	!Check that there are no more than 3 numbers in the signal description
	WHILE n_CharNumberCount>2 DO
		TPErase;
		st_MsgBoxHeader:=["GetGOValue  Signal=" + st_doSignalName ,"GetGOValue  Signal=" + st_doSignalName,"???"];
		st_MsgBoxLine3:=["There are more than two numbers in the" ,"Es gibt mehr als zwei Zahlen in der","???"];
		st_MsgBoxLine4:=["signal name defined. Check Configuration.","Signal-Name definiert. Konfiguration prüfen.","???"];
		n_MsgBoxAnswer:= UIMessageBox (\Header:=st_MsgBoxHeader{n_Sp}\MsgArray:=[" "," ",st_MsgBoxLine3{n_Sp},st_MsgBoxLine4{n_Sp}," "]\Buttons:=btnOK\Icon:=iconError) ;

		STOP;
	ENDWHILE

	!Check that there are no less than numbers in signal description
	WHILE n_CharNumberCount<2 DO
		TPErase;
		st_MsgBoxHeader:=["GetGOValue  Signal=" + st_doSignalName ,"GetGOValue  Signal=" + st_doSignalName,"???"];
		st_MsgBoxLine3:=["The are less than two numbers in the" ,"???","???"];
		st_MsgBoxLine4:=["signal name defined. Check Configuration.","Signal-Name definiert. Konfiguration prüfen.","???"];
		n_MsgBoxAnswer:= UIMessageBox (\Header:=st_MsgBoxHeader{n_Sp}\MsgArray:=[" "," ",st_MsgBoxLine3{n_Sp},st_MsgBoxLine4{n_Sp}," "]\Buttons:=btnOK\Icon:=iconError) ;

		STOP;
	ENDWHILE

	!Get Bit number as a string
	st_FirstbitNr:=StrPart(st_doSignalName,n_CharFirstNumber,n_NumberCharlength);

	!Check st_FirstbitNr is a number
	WHILE StrToVal(st_FirstbitNr,n_FirstBitNr)<>TRUE DO
		TPErase;
		st_MsgBoxHeader:=["GetGOValue  Signal=" + st_doSignalName ,"GetGOValue  Signal=" + st_doSignalName,"???"];
		st_MsgBoxLine3:=["There are not two consecutive bit numbers defined." ,"Es gibt nicht zwei aufeinander folgenden Bit-Zahlen definiert.","???"];
		st_MsgBoxLine4:=["Please Check Configuration.","Bitte Überprüfe Konfiguration.","???"];
		n_MsgBoxAnswer:= UIMessageBox (\Header:=st_MsgBoxHeader{n_Sp}\MsgArray:=[" "," ",st_MsgBoxLine3{n_Sp},st_MsgBoxLine4{n_Sp}," "]\Buttons:=btnOK\Icon:=iconError) ;

		STOP;
	ENDWHILE

	st_doSignalDesc1:=StrPart(st_doSignalName,1,n_CharFirstNumber-1);

	IF (n_CharFirstNumber+1)=n_doSignal_Length OR n_CharFirstNumber=n_doSignal_Length THEN
		!Bit numbers are the last two characters
		st_doSignalDesc2:="" ;
		st_doSignalDesc:=st_doSignalDesc1 + "??" ;
	ELSE
		st_doSignalDesc2:=StrPart(st_doSignalName,n_CharFirstNumber+2,n_doSignal_Length-n_CharFirstNumber-1);
		st_doSignalDesc:=st_doSignalDesc1 + "??" + st_doSignalDesc2 ;
	ENDIF

	n_LastBitNr:=n_FirstBitNr+n_doBitLength-1;

	IF n_doBitLength<1 OR n_doBitLength>16 THEN
		!Check n_doBitLength paramater is valid

		WHILE TRUE DO
			TPErase;
			st_MsgBoxHeader:=["GetGOValue  Signal=" + st_doSignalName ,"GetGOValue  Signal=" + st_doSignalName,"???"];
			st_MsgBoxLine3:=["The Bit length Specified=" + ValToStr(n_doBitLength) + ". Value must be between 1-16." ,"Die Bitlänge angegeben=" + ValToStr(n_doBitLength) + ". Wert muss zwischen 1-16.","???"];
			st_MsgBoxLine4:=["Please Check Configuration.","Bitte Überprüfe Konfiguration.","???"];
			n_MsgBoxAnswer:= UIMessageBox (\Header:=st_MsgBoxHeader{n_Sp}\MsgArray:=[" "," ",st_MsgBoxLine3{n_Sp},st_MsgBoxLine4{n_Sp}," "]\Buttons:=btnOK\Icon:=iconError) ;

			STOP;
		ENDWHILE

	ELSEIF n_LastBitNr>32 THEN
		!Check last bit number

		WHILE TRUE DO
			TPErase;
			st_MsgBoxHeader:=["GetGOValue  Signal=" + st_doSignalName ,"GetGOValue  Signal=" + st_doSignalName,"???"];
			st_MsgBoxLine3:=["The first Bit specified=" + ValToStr(n_FirstBitNr) + " + length specified=" + ValToStr(n_doBitLength) + " is >32.","Die Erstes Bit angegeben=" + ValToStr(n_FirstBitNr) + " + Länge angegeben=" + ValToStr(n_doBitLength) + " ist >32.","???"];
			st_MsgBoxLine4:=["Please Check Configuration.","Bitte Überprüfe Konfiguration.","???"];
			n_MsgBoxAnswer:= UIMessageBox (\Header:=st_MsgBoxHeader{n_Sp}\MsgArray:=[" "," ",st_MsgBoxLine3{n_Sp},st_MsgBoxLine4{n_Sp}," "]\Buttons:=btnOK\Icon:=iconError) ;

			STOP;
		ENDWHILE

	ELSE !n_doBitLength<1
		n_ScrollNr:=0.5;
		n_ValueCount:=0;

		FOR n_CharNr FROM n_FirstBitNr	TO n_LastBitNr DO
			n_ScrollNr:=n_ScrollNr*2;

			IF n_CharNr<10 AND n_CharFirstNumber<>n_doSignal_Length THEN
				st_tempString:=st_doSignalDesc1 +"0" + ValToStr(n_CharNr) + st_doSignalDesc2;
			ELSE
				st_tempString:=st_doSignalDesc1 + ValToStr(n_CharNr) + st_doSignalDesc2;
			ENDIF

			AliasIO st_tempString, do_Temp;

			IF doutput(do_Temp) = 1 THEN
				n_ValueCount:=n_ValueCount + n_ScrollNr ;
			ENDIF

		ENDFOR

		n_LastGroupOutput:=n_ValueCount;
		RETURN n_ValueCount ;
	ENDIF !n_doBitLength<1
ENDIF !n_diSignal_Length

ERROR
!** Error Handler **

TEST  ERRNO
CASE ERR_ALIASIO_DEF,ERR_ALIASIO_TYPE :
	WHILE TRUE DO
		TPErase;
		st_MsgBoxHeader:=["GetGOValue Signal=" + st_tempString ,"GetGOValue Signal=" + st_tempString,"???"];
		st_MsgBoxLine3:=["Signal is missing or incorrectly defined","IO Signal ist nicht vorhanden oder Falsch geschrieben","???"];
		st_MsgBoxLine4:=["Please Check Configuration.","Bitte Überprüfe Konfiguration.","???"];
		n_MsgBoxAnswer:= UIMessageBox (\Header:=st_MsgBoxHeader{n_Sp}\MsgArray:=[" "," ",st_MsgBoxLine3{n_Sp},st_MsgBoxLine4{n_Sp}," "]\Buttons:=btnOK\Icon:=iconError) ;

		STOP;
	ENDWHILE
DEFAULT :
	WHILE TRUE DO
		TPErase;
		st_MsgBoxHeader:=["GetGOValue Unknown Error =" + ValToStr(Errno) ,"GetGOValue unbekannter Fehler =" + ValToStr(Errno),"???"];
		st_MsgBoxLine3:=["Support Required.","Unterstützung erforderlich.","???"];
		st_MsgBoxLine4:=[" "," ","???"];
		n_MsgBoxAnswer:= UIMessageBox (\Header:=st_MsgBoxHeader{n_Sp}\MsgArray:=[" "," ",st_MsgBoxLine3{n_Sp},st_MsgBoxLine4{n_Sp}," "]\Buttons:=btnOK\Icon:=iconError) ;

		STOP;
	ENDWHILE
ENDTEST

ENDFUNC !(GetGroupOP)


!*******************************************************************************


PROC SetGroupOP (VAR Signaldo doSignalName,Num n_doBitLength,Num n_doSetValue)
!************************************
!* Procedure set a group of Digital *
!* Outputs based on a numeric value *
!************************************

VAR signaldo do_Temp;

VAR Byte by_HighByte ;
VAR Byte by_LowByte ;
VAR Byte by_BitMask;

VAR Num n_FirstBitNr;
VAR Num n_LastBitNr;
VAR Num n_doSignal_Length;
VAR Num n_CharNr;
VAR Num n_ScrollNr;
VAR Num n_CharFirstNumber;
VAR Num n_CharNumberCount;
VAR Num n_MaxValue ;
VAR Num n_TempNr ;
VAR Num n_ChkValue ;
VAR Num n_TempDoValue ;

VAR String st_doSignalName;
VAR String st_FirstbitNr;
VAR String st_doSignalDesc;
VAR String st_doSignalDesc1;
VAR String st_doSignalDesc2;
VAR String st_tempString ;

!Stop advance pointer
WaitTime\Inpos, 0.0 ;

!Check first bit configured is a valid output
st_doSignalName:=ArgName(doSignalName);
AliasIO st_doSignalName, do_Temp;

!Check output name length
n_doSignal_Length:=StrLen(st_doSignalName);

IF n_doSignal_Length > 3 THEN
	!Determine which characters the Bit numbers start
	n_CharFirstNumber:=StrFind(st_doSignalName,1,STR_DIGIT) ;

	!Check that there are numbers in signal description
	WHILE n_CharFirstNumber>n_doSignal_Length DO
		TPErase;
		st_MsgBoxHeader:=["SetGOValue Signal=" + st_doSignalName ,"SetGOValue Signal=" + st_doSignalName,"???"];
		st_MsgBoxLine3:=["There are no bit numbers in the signal name defined." ,"Es gibt keine Bit-Zahlen in der Signal-Namen definiert","???"];
		st_MsgBoxLine4:=["Please Check Configuration.","Bitte Überprüfe Konfiguration.","???"];
		n_MsgBoxAnswer:= UIMessageBox (\Header:=st_MsgBoxHeader{n_Sp}\MsgArray:=[" "," ",st_MsgBoxLine3{n_Sp},st_MsgBoxLine4{n_Sp}," "]\Buttons:=btnOK\Icon:=iconError) ;

		STOP;
	ENDWHILE

	n_CharNumberCount:=1;

	!Check how many characters are numbers
	FOR n_CharNr FROM n_CharFirstNumber +1 TO n_doSignal_Length DO
		IF StrFind(st_doSignalName,n_CharNr,STR_DIGIT)<=n_doSignal_Length THEN
			INCR n_CharNumberCount ;
		ENDIF
	ENDFOR

	!Check that there are no more than 3 numbers in the signal description
	WHILE n_CharNumberCount>2 DO
		TPErase;
		st_MsgBoxHeader:=["SetGOValue Signal=" + st_doSignalName ,"SetGOValue Signal=" + st_doSignalName,"???"];
		st_MsgBoxLine3:=["There are more than two numbers in the" ,"Es gibt mehr als zwei Zahlen in der","???"];
		st_MsgBoxLine4:=["signal name defined. Check Configuration.","Signal-Name definiert. Konfiguration prüfen.","???"];
		n_MsgBoxAnswer:= UIMessageBox (\Header:=st_MsgBoxHeader{n_Sp}\MsgArray:=[" "," ",st_MsgBoxLine3{n_Sp},st_MsgBoxLine4{n_Sp}," "]\Buttons:=btnOK\Icon:=iconError) ;

		STOP;
	ENDWHILE

	!Check that there are no less than numbers in signal description
	WHILE n_CharNumberCount<2 DO
		TPErase;
		st_MsgBoxHeader:=["SetGOValue Signal=" + st_doSignalName ,"SetGOValue Signal=" + st_doSignalName,"???"];
		st_MsgBoxLine3:=["The are less than two numbers in the" ,"???","???"];
		st_MsgBoxLine4:=["signal name defined. Check Configuration.","Signal-Name definiert. Konfiguration prüfen.","???"];
		n_MsgBoxAnswer:= UIMessageBox (\Header:=st_MsgBoxHeader{n_Sp}\MsgArray:=[" "," ",st_MsgBoxLine3{n_Sp},st_MsgBoxLine4{n_Sp}," "]\Buttons:=btnOK\Icon:=iconError) ;

		STOP;
	ENDWHILE

	!Get Bit number as a string
	st_FirstbitNr:=StrPart(st_doSignalName,n_CharFirstNumber,2);

	!Check st_FirstbitNr is a number
	WHILE StrToVal(st_FirstbitNr,n_FirstBitNr)<>TRUE DO
		TPErase;
		st_MsgBoxHeader:=["SetGOValue Signal=" + st_doSignalName ,"SetGOValue Signal=" + st_doSignalName,"???"];
		st_MsgBoxLine3:=["There are not two consecutive bit numbers defined." ,"Es gibt nicht zwei aufeinander folgenden Bit-Zahlen definiert.","???"];
		st_MsgBoxLine4:=["Please Check Configuration.","Bitte Überprüfe Konfiguration.","???"];
		n_MsgBoxAnswer:= UIMessageBox (\Header:=st_MsgBoxHeader{n_Sp}\MsgArray:=[" "," ",st_MsgBoxLine3{n_Sp},st_MsgBoxLine4{n_Sp}," "]\Buttons:=btnOK\Icon:=iconError) ;

		STOP;
	ENDWHILE

	st_doSignalDesc1:=StrPart(st_doSignalName,1,n_CharFirstNumber-1);

	IF (n_CharFirstNumber+1)=n_doSignal_Length THEN
		!Bit numbers are the last two characters
		st_doSignalDesc2:="" ;
		st_doSignalDesc:=st_doSignalDesc1 + "??" ;
	ELSE
		st_doSignalDesc2:=StrPart(st_doSignalName,n_CharFirstNumber+2,n_doSignal_Length-n_CharFirstNumber-1);
		st_doSignalDesc:=st_doSignalDesc1 + "??" + st_doSignalDesc2 ;
	ENDIF

	n_LastBitNr:=n_FirstBitNr+n_doBitLength-1;

	IF n_doBitLength<1 OR n_doBitLength>16 THEN
		!Check n_doBitLength paramater is valid

		WHILE TRUE DO
			TPErase;
			st_MsgBoxHeader:=["SetGOValue Signal=" + st_doSignalName ,"SetGOValue Signal=" + st_doSignalName,"???"];
			st_MsgBoxLine3:=["The Bit length Specified=" + ValToStr(n_doBitLength) + ". Value must be between 1-16." ,"Die Bitlänge angegeben=" + ValToStr(n_doBitLength) + ". Wert muss zwischen 1-16.","???"];
			st_MsgBoxLine4:=["Please Check Configuration.","Bitte Überprüfe Konfiguration.","???"];
			n_MsgBoxAnswer:= UIMessageBox (\Header:=st_MsgBoxHeader{n_Sp}\MsgArray:=[" "," ",st_MsgBoxLine3{n_Sp},st_MsgBoxLine4{n_Sp}," "]\Buttons:=btnOK\Icon:=iconError) ;

			STOP;
		ENDWHILE

	ELSEIF n_LastBitNr>32 THEN
		!Check last bit number

		WHILE TRUE DO
			TPErase;
			st_MsgBoxHeader:=["SetGOValue Signal=" + st_doSignalName ,"SetGOValue Signal=" + st_doSignalName,"???"];
			st_MsgBoxLine3:=["The first Bit specified=" + ValToStr(n_FirstBitNr) + " + length specified=" + ValToStr(n_doBitLength) + " is >32.","Die Erstes Bit angegeben=" + ValToStr(n_FirstBitNr) + " + Länge angegeben=" + ValToStr(n_doBitLength) + " ist >32.","???"];
			st_MsgBoxLine4:=["Please Check Configuration.","Bitte Überprüfe Konfiguration.","???"];
			n_MsgBoxAnswer:= UIMessageBox (\Header:=st_MsgBoxHeader{n_Sp}\MsgArray:=[" "," ",st_MsgBoxLine3{n_Sp},st_MsgBoxLine4{n_Sp}," "]\Buttons:=btnOK\Icon:=iconError) ;

			STOP;
		ENDWHILE

	ELSE !n_doBitLength<1

		!Calculate maximum value allowed
		n_MaxValue:=0.5;

		FOR n_TempNr FROM n_FirstBitNr	TO n_LastBitNr +1 DO
			n_MaxValue:=n_MaxValue*2;
		ENDFOR

		Decr n_MaxValue ;

		!Check value number enterd is a permitted value
		WHILE n_doSetValue<0 OR n_doSetValue>n_MaxValue DO
			TPErase;
			st_MsgBoxHeader:=["SetGOValue Signal=" + st_doSignalName ,"SetGOValue Signal=" + st_doSignalName,"???"];
			st_MsgBoxLine3:=["The Group Output value set=" + ValToStr(n_doSetValue) ,"Der Konzern Ausgangswert eingestellt=" + ValToStr(n_doSetValue),"???"];
			st_MsgBoxLine4:=["It must be a value between 0-" + ValToStr(n_MaxValue) +". Check Configuration.","Es muss ein Wert zwischen sein 0-" + ValToStr(n_MaxValue) +". überprüfen Konfiguration.","???"];
			n_MsgBoxAnswer:= UIMessageBox (\Header:=st_MsgBoxHeader{n_Sp}\MsgArray:=[" "," ",st_MsgBoxLine3{n_Sp},st_MsgBoxLine4{n_Sp}," "]\Buttons:=btnOK\Icon:=iconError) ;

			STOP;
		ENDWHILE

		!Set Low & High byte
		by_LowByte:=0 ;
		by_HighByte:=0 ;
		n_ChkValue:=32768 ;
		n_TempDoValue:=n_doSetValue ;

		FOR n_TempNr FROM 16 TO 1 STEP -1 DO
			IF n_TempDoValue>=n_ChkValue THEN
				n_TempDoValue:=n_TempDoValue-n_ChkValue ;

				IF n_TempNr>8 THEN
					!Set High Byte
					BitSet by_HighByte, n_TempNr-8;
				ELSE
					!Set Low Byte
					BitSet by_LowByte, n_TempNr;
				ENDIF
			ENDIF

			n_ChkValue:=n_ChkValue-(n_ChkValue/2) ;
		ENDFOR

		!Set Outputs control
		n_ScrollNr:=0;

		FOR n_TempNr FROM n_FirstBitNr	TO n_LastBitNr DO
			Incr n_ScrollNr ;

			IF n_ScrollNr=1 OR n_ScrollNr=9 THEN
				by_BitMask:=1;
			ELSE
				by_BitMask:=by_BitMask*2 ;
			ENDIF

 			IF n_TempNr<10 THEN
				st_tempString:=st_doSignalDesc1 +"0" + ValToStr(n_TempNr) + st_doSignalDesc2;
			ELSE
				st_tempString:= st_doSignalDesc1 + ValToStr(n_TempNr) + st_doSignalDesc2;
			ENDIF

			AliasIO st_tempString, do_Temp;

			IF n_ScrollNr<9 THEN
				!Low Byte
				B_Setdo do_Temp,(BitAND(by_LowByte,by_BitMask)<>0) ;
			ELSE
				!High Byte
				B_Setdo do_Temp,(BitAND(by_HighByte,by_BitMask)<>0) ;
			ENDIF
		ENDFOR
	ENDIF !n_doBitLength<1
ENDIF !n_doSignal_Length

ERROR
!** Error Handler **

TEST  ERRNO
CASE ERR_ALIASIO_DEF,ERR_ALIASIO_TYPE :
	WHILE TRUE DO
		TPErase;
		st_MsgBoxHeader:=["SetGOValue Signal=" + st_tempString ,"SetGOValue Signal=" + st_tempString,"???"];
		st_MsgBoxLine3:=["Signal is missing or incorrectly defined","IO Signal ist nicht vorhanden oder Falsch geschrieben","???"];
		st_MsgBoxLine4:=["Please Check Configuration.","Bitte Überprüfe Konfiguration.","???"];
		n_MsgBoxAnswer:= UIMessageBox (\Header:=st_MsgBoxHeader{n_Sp}\MsgArray:=[" "," ",st_MsgBoxLine3{n_Sp},st_MsgBoxLine4{n_Sp}," "]\Buttons:=btnOK\Icon:=iconError) ;

		STOP;
	ENDWHILE

DEFAULT :

	WHILE TRUE DO
		TPErase;
		st_MsgBoxHeader:=["SetGOValue Unknown Error =" + ValToStr(Errno) ,"SetGOValue unbekannter Fehler =" + ValToStr(Errno),"???"];
		st_MsgBoxLine3:=["Support Required.","Unterstützung erforderlich.","???"];
		st_MsgBoxLine4:=[" "," ","???"];
		n_MsgBoxAnswer:= UIMessageBox (\Header:=st_MsgBoxHeader{n_Sp}\MsgArray:=[" "," ",st_MsgBoxLine3{n_Sp},st_MsgBoxLine4{n_Sp}," "]\Buttons:=btnOK\Icon:=iconError) ;

		STOP;
	ENDWHILE
ENDTEST

ENDPROC !(SetGroupOP)


!*******************************************************************************


PROC CheckManualTestMode ()
!**********************************
!* Procedure To check Mode switch *
!*  is switched to Manual (Slow)  *
!**********************************
VAR ErrNum en_DO_Break;

WHILE (OpMode()<>OP_MAN_PROG) DO
	TPErase;
	st_MsgBoxHeader:=["Check Mode Keyswitch" ,"Check Mode Keyswitch","???"];
	st_MsgBoxLine3:=["This progam may only be called","Das Progamm kann nur aufgerufen werden","???"];
	st_MsgBoxLine4:=["in Manual Prog (Slow) 'T1' mode.","im Manual Prog (Slow) 'T1'-Modus.","???"];
	n_MsgBoxAnswer:= UIMessageBox (\Header:=st_MsgBoxHeader{n_Sp}\MsgArray:=[" "," ",st_MsgBoxLine3{n_Sp},st_MsgBoxLine4{n_Sp}," "]\Buttons:=btnOK\Icon:=iconError\DoBreak:=SYS_do_Manual\BreakFlag:=en_DO_Break) ;

	STOP;
ENDWHILE

ENDPROC !(CheckManualTestMode)


!*******************************************************************************


PROC B_Setdo (VAR signaldo do_Output,BOOL State)
!******************************************
!* Procedure To work with Digital Outputs *
!* as if they were  declared as a Boolean *
!******************************************

IF State THEN
	SET do_Output;
ELSE
	RESET do_Output;
ENDIF

ENDPROC !(B_SetOut)


!*******************************************************************************


FUNC Num GetTypeCode ()
!*********************************
!* Function to return a numeric  *
!*   code from type bits 1-10    *
!*  providing only one bit is on *
!*********************************

VAR Signaldi di_Temp;
VAR String st_diSignalName;
VAR Num n_ReturnValue:=0;

FOR i FROM 1 TO 10 DO
	IF i<10 THEN
		st_diSignalName:="PLC_di_Typbit_0" + ValToStr(i);
	ELSE
		st_diSignalName:="PLC_di_Typbit_10";
	ENDIF

	AliasIO st_diSignalName, di_Temp;

	IF di_Temp = 1 THEN
		IF  n_ReturnValue=0 THEN
			n_ReturnValue:=i;
		ELSE
			n_ReturnValue:=0;
			GOTO ExitFor ;
		ENDIF
	ENDIF

ENDFOR

ExitFor:

RETURN n_ReturnValue;

ENDFUNC !(GetTypeCode)


!*******************************************************************************


PROC SetTypeCode (Num n_CodeValue)
!*********************************
!*   Procedure to set a model    *
!*   code with type bits 1-10    *
!*         to the PLC            *
!*********************************

VAR Signaldo do_Temp;
VAR String st_doSignalName;

CheckValue n_CodeValue, 1, 10, 0, "SetTypeCode";

FOR i FROM 1 TO 10 DO
	IF i<10 THEN
		st_doSignalName:="PLC_do_Typbit_0" + ValToStr(i);
	ELSE
		st_doSignalName:="PLC_do_Typbit_10";
	ENDIF

	AliasIO st_doSignalName, do_Temp;

	IF i=n_CodeValue AND n_CodeValue>0 AND n_CodeValue<=10 THEN
		SET do_Temp ;
	ELSE
		RESET do_Temp ;
	ENDIF

ENDFOR

ENDPROC !(SetTypeCode)
!***************************************************************************

PROC SetRobotTypeCode (\ Num GripperSystem,\ Bool PartOnGripper,\Switch InPos )
!******************************************************
!* Procedure to set a Robot Type code Bits to the PLC *
!*       depending upon gripper system selected       *
!******************************************************

VAR Signaldo do_Temp;
VAR String st_doSignalName;
VAR Num n_Offset;

! Only execute function if optional arguments are used and a valid gripper system number is entered
IF Present (GripperSystem) AND  Present (PartOnGripper) THEN

	CheckValue GripperSystem, 1, 4, 0, "SetRobotTypeCode";

	IF Present(InPos) THEN
		WaitTime \Inpos,0;
		!***********************************
		! Waiting for robot motion pointer *
		!***********************************
	ENDIF

	n_Offset:=(GripperSystem*2)-1;

	st_doSignalName:="PLC_do_Typbit_" + ValToStr(24+n_Offset);
	AliasIO st_doSignalName, do_Temp;

	B_Setdo do_Temp,PartOnGripper;

	st_doSignalName:="PLC_do_Typbit_" + ValToStr(25+n_Offset);
	AliasIO st_doSignalName, do_Temp;

	B_Setdo do_Temp,NOT PartOnGripper;

ENDIF

ENDPROC !(SetRobotTypeCode)

!***************************************************************************

PROC Indirect_WOBJ(tooldata Mess_Tool,INOUT wobjdata Wobj_New)
!***********************************
!*   Define Indirect Work Object   *
!***********************************
VAR num n_key;
VAR pose Punkt;
VAR pose u_pose;
VAR num n_ErrorCode;
VAR bool M_Errror;

!Update Phil Parsons 16-June-2012

Begin:
M_Errror:=FALSE;
n_ErrorCode:=0;

t_DefWobj_Act_tool:=Mess_Tool;

s_DefWobj_Tool_Name:=ArgName(Mess_Tool);
s_DefWobj_Wobj_Name:=ArgName(Wobj_New);

IF IsPers(Wobj_New)=FALSE THEN
	TPErase;
	TEST n_sp
	CASE 1:
		TPWrite "The workobject "+s_DefWobj_Wobj_Name;
		TPWrite "is incorrectly declared.";
		TPWrite "----------------------------------------";
		TPWrite "It must be declared as a type 'PERS'.";
	CASE 2:
	    TPWrite "Das uebergebene Werkobjekt "+s_DefWobj_Wobj_Name;
		TPWrite "ist nicht vom Typ SPEICHERND ";
		TPWrite "----------------------------------------";
		TPWrite "Variable muss umdeklariert werden!";
	CASE 3:

	ENDTEST

	TPReadFK n_key,"","","","","","OK";

	GOTO Exit_Ende;
ENDIF

TPErase;
TEST n_sp
CASE 1:
	TPWrite "Work object defined using  ";
	TPWrite "3 measurement points ";
	TPWrite "----------------------------------------";
	TPWrite "The Work Object name is "+s_DefWobj_Wobj_Name ;
	TPWrite "using measurement tool "+s_DefWobj_Tool_Name ;
	TPReadFK n_key,"","Abort","","","","OK";
CASE 2:
	TPWrite "Werkobjektdefinition mit Hilfe von  ";
    TPWrite "3 Punkten vermessen im Werkobjekt   ";
    TPWrite "----------------------------------------";
    TPWrite "Es wird das Werkobjekt "+s_DefWobj_Wobj_Name;
    TPWrite "mit Hilfe des Mess-Tool "+s_DefWobj_Tool_Name;
    TPWrite "bestimmt!";
    TPReadFK n_key,"","Abbruch","","","","OK";
CASE 3:

ENDTEST

IF n_key=1 GOTO Exit_Ende;

IF n_key<>5 GOTO Begin;

WHILE CTool()<>t_DefWobj_Act_tool DO
 	 TPErase;

	TEST n_sp
	CASE 1:
		TPWrite "               WARNING!!  ";
		TPWrite "----------------------------------------";
		TPWrite "The current Tool used to Jog ";
		TPWrite "is not the measurement tool "+s_DefWobj_Tool_Name;
 		TPReadFK n_key,"Please change the jogging tool !","Abort","","","","OK";
	CASE 2:
		TPWrite "               ACHTUNG !  ";
		TPWrite "----------------------------------------";
		TPWrite "Das im Bewegenfenster eingestellte ";
		TPWrite "TOOL ist nicht gleich dem angegebenen";
		TPWrite "Mess-TOOL "+s_DefWobj_Tool_Name;
		TPReadFK n_key,"Muss geaendet werden!","Abbruch","","","","OK";
	CASE 3:

	ENDTEST

  	IF n_key=1 GOTO Exit_Ende;
ENDWHILE

FOR I FROM 1 TO 3 DO
	Re_Start:
	TPErase;

	TEST n_sp
	CASE 1:
		TPWrite "What do you want to do with measurement point" + NumToStr(I,0)+ " ?";
		TPWrite " ";
		TPWrite " - Teach new.";
		TPWrite " - Change exiting data.";
		TPWrite " - Move the robot to the point.";
		TPWrite "";
		TPReadFK n_key,"Please select option.","Teach New","","Change","","Goto Point";
	CASE 2:
		TPWrite "Wollen Sie Mess-Punkt" + NumToStr(I,0)+ " ?";
		TPWrite " ";
		TPWrite " - neu teachen";
		TPWrite " - gespeicherten Mess-Punkt uebernehmen";
		TPWrite " - gespeicherten Punkt anfahren und ggf.";
		TPWrite "   korrigieren";
		TPWrite "";
		TPReadFK n_key,"Bitte wählen Sie Option.","teachen","","uebernahme","","anfahren";
	CASE 3:

	ENDTEST

	TEST n_key
	CASE 1:
		GOTO Teach;
	CASE 3:
		GOTO Posexyz;
	CASE 5:
		GOTO ToPoint;
	DEFAULT:
		GOTO Re_Start;
	ENDTEST

	ToPoint:
	WHILE OpMode()<>2 DO
		TPErase;

		TEST n_sp
		CASE 1:
			TPWrite "              WARNING!                  ";
			TPWrite "----------------------------------------";
			TPWrite "This program may only be run in Manual ";
			TPWrite "program 'T1' mode.";
			TPReadFK n_key,"Please Turn the Key switch to manual!","Abort","","","","OK";
		CASE 2:
			TPWrite "              ACHTUNG!                  ";
			TPWrite "----------------------------------------";
			TPWrite "Bewegungsart ist nicht auf Hand-Betrieb!";
			TPWrite "Anfahren des Mess-Punktes ist nur in";
			TPWrite "dieser Betriebs-Art möglich!";
			TPReadFK n_key,"Stellen Sie auf Betriebs-Art Hand um!","Abbruch","","","","OK";
		CASE 3:

		ENDTEST

		IF n_key=1 GOTO Exit_Ende;
	ENDWHILE

	TPErase;

	TEST n_sp
	CASE 1:

		TPWrite "      WARNING!  RICK OF COLLISION !     ";
		TPWrite "----------------------------------------";
		TPWrite "The Robot will move directly to the ";
		TPWrite "previously stored measurement point "\Num:=I;
		TPReadFK n_key,"","Return","","","Move Fast","Move Slow";
	CASE 2:
		TPWrite "     ACHTUNG!     KOLLISIONSGEFAHR!     ";
		TPWrite "----------------------------------------";
		TPWrite "Roboter bewegt sich auf direktem Wege";
		TPWrite "zum gespeichertem Mess-Punkt "\Num:=I;
		TPReadFK n_key,"","Zurueck","","","schnell","langsam";
	CASE 3:

	ENDTEST

	TPErase;

	TEST n_key
	CASE 1:
		GOTO Re_Start;
	CASE 4:
		n_ErrorCode:=1;
		MoveJ rt_DefWobj_user_p{I},vmax,fine,t_DefWobj_Act_tool;
		n_ErrorCode:=0;
	CASE 5:
		n_ErrorCode:=1;
		MoveJ rt_DefWobj_user_p{I},v50,fine,t_DefWobj_Act_tool;
		n_ErrorCode:=0;
	DEFAULT:
		GOTO Re_Start;
	ENDTEST

	Teach:
	TPErase;

	TEST n_sp
	CASE 1:
		TPWrite "Jog the robot to the measurement ";
		TPWrite "point with the tool "+s_DefWobj_Tool_Name+".";
		TPWrite "The current Measurement Point is "\Num:=I;
		TPReadFK n_key,"Has the point been Reached?","Return","","","","Yes";
	CASE 2:
		TPWrite "Bewegen Sie den Roboter mit dem ";
		TPWrite "Mess-Werkzeug "+s_DefWobj_Tool_Name+" zum";
		TPWrite "vermessenen Punkt "\Num:=I;
		TPReadFK n_key,"Ist der Punkt erreicht?","Zurueck","","","","Ja";
	CASE 3:

	ENDTEST

	IF n_key=1 GOTO Re_Start;
	IF n_key<>5 GOTO teach;

	rt_DefWobj_user_p{I}:=CRobT(\Tool:=t_DefWobj_Act_tool\WObj:=wobj0);

	Posexyz:
	TPErase;

	TEST n_sp
	CASE 1:
		TPWrite "The Co-Ordinates for measurement point "\Num:=I;
		TPWrite "for this Work Object are:";
		TPWrite " ";
		TPWrite "   X=: "\Num:=rt_DefWobj_mess_p{I}.trans.x;
		TPWrite "   Y=: "\Num:=rt_DefWobj_mess_p{I}.trans.y;
		TPWrite "   Z=: "\Num:=rt_DefWobj_mess_p{I}.trans.z;
		TPWrite " ";
		TPReadFK n_key,"Are The Co-Ordinates correct?","No","","","","Yes";
	CASE 2:
		TPWrite "Die Koordinaten fuer Mess-Punkt "\Num:=I;
		TPWrite "im Bezug zum Werkobjekt sind:";
		TPWrite " ";
		TPWrite "   X-Wert: "\Num:=rt_DefWobj_mess_p{I}.trans.x;
		TPWrite "   Y-Wert: "\Num:=rt_DefWobj_mess_p{I}.trans.y;
		TPWrite "   Z-Wert: "\Num:=rt_DefWobj_mess_p{I}.trans.z;
		TPWrite " ";
		TPReadFK n_key,"Sind die Koordinaten richtig?","Nein","","","","Ja";
	CASE 3:

	ENDTEST

	IF n_key=5 GOTO Pose_ok;
	New_Pos:
	n_DefWobj_px:=0;
	n_DefWobj_py:=0;
	n_DefWobj_pz:=0;
	TPErase;

	TEST n_sp
	CASE 1:
		TPWrite "Manually enter ";
		TPWrite "the Co-Ordinates ";
		TPWrite "for the Work Object!";
		TPWrite "for point "\Num:=I;
		TPReadNum n_DefWobj_px,"X-Value:";
		TPErase;
		TPWrite "Manually enter ";
		TPWrite "the Co-Ordinates ";
		TPWrite "for the Work Object!";
		TPWrite "for point "\Num:=I;
		TPReadNum n_DefWobj_py,"Y-Value:";
		TPErase;
		TPWrite "Manually enter ";
		TPWrite "the Co-Ordinates ";
		TPWrite "for the Work Object!";
		TPWrite "for point "\Num:=I;
		TPReadNum n_DefWobj_pz,"Z-Value:";
	CASE 2:
		TPWrite "Geben Sie per Hand die ";
		TPWrite "Koordinaten des Punktes ";
		TPWrite "zum Werkobjekt ein!";
		TPWrite "Punkt "\Num:=I;
		TPReadNum n_DefWobj_px,"X-Wert:";
		TPErase;
		TPWrite "Geben Sie per Hand die ";
		TPWrite "Koordinaten des Punktes ";
		TPWrite "zum Werkobjekt ein!";
		TPWrite "Punkt "\Num:=I;
		TPReadNum n_DefWobj_py,"Y-Wert:";
		TPErase;
		TPWrite "Geben Sie per Hand die ";
		TPWrite "Koordinaten des Punktes ";
		TPWrite "zum Werkobjekt ein!";
		TPWrite "Punkt "\Num:=I;
 		TPReadNum n_DefWobj_pz,"Z-Wert:";
	CASE 3:

	ENDTEST

	Pose_frag:
	TPErase;

	TEST n_sp
	CASE 1:
		TPWrite "The value entered for measurement point "\Num:=I;
		TPWrite "are for the Work Object:";
		TPWrite " ";
		TPWrite "   X-Value: "\Num:=n_DefWobj_px;
		TPWrite "   Y-Value: "\Num:=n_DefWobj_py;
		TPWrite "   Z-Value: "\Num:=n_DefWobj_pz;
		TPWrite " ";
		TPReadFK n_key,"Are the Co-Ordinates correct?","No","","Abort","","Yes";
	CASE 2:
		TPWrite "Die eingegebenen Werte fuer Mess-Punkt "\Num:=I;
		TPWrite "im Bezug zum Werkobjekt sind:";
		TPWrite " ";
		TPWrite "   X-Wert: "\Num:=n_DefWobj_px;
		TPWrite "   Y-Wert: "\Num:=n_DefWobj_py;
		TPWrite "   Z-Wert: "\Num:=n_DefWobj_pz;
		TPWrite " ";
		TPReadFK n_key,"Sind die Koordinaten richtig?","Nein","","","","Ja";
	CASE 3:

	ENDTEST

	IF n_key=3 GOTO Exit_Ende;
	IF n_key=1 GOTO New_Pos;
	IF n_key<>5 GOTO Pose_frag;

	rt_DefWobj_mess_p{I}.trans.x:=n_DefWobj_px;
	rt_DefWobj_mess_p{I}.trans.y:=n_DefWobj_py;
	rt_DefWobj_mess_p{I}.trans.z:=n_DefWobj_pz;
	rt_DefWobj_mess_p{I}.rot:=[1,0,0,0];
	Pose_ok:
ENDFOR

TPErase;
n_ErrorCode:=2;
wobj_DefWobj_car0.oframe:=[[0,0,0],[1,0,0,0]];
wobj_DefWobj_car0.uframe:=DefDFrame(rt_DefWobj_mess_p{1},rt_DefWobj_mess_p{2},rt_DefWobj_mess_p{3},rt_DefWobj_user_p{1},rt_DefWobj_user_p{2},rt_DefWobj_user_p{3});
IF M_Errror=TRUE GOTO Ende;
n_ErrorCode:=0;

FOR I FROM 1 TO 3 DO
	Punkt.trans:=rt_DefWobj_mess_p{I}.trans;
	Punkt.rot:=rt_DefWobj_mess_p{I}.rot;
	u_pose:=PoseMult(wobj_DefWobj_car0.uframe,Punkt);
	n_DefWobj_Diff_X{I}:=u_pose.trans.x-rt_DefWobj_user_p{I}.trans.x;
	n_DefWobj_Diff_Y{I}:=u_pose.trans.y-rt_DefWobj_user_p{I}.trans.y;
	n_DefWobj_Diff_Z{I}:=u_pose.trans.z-rt_DefWobj_user_p{I}.trans.z;
	n_DefWob_jDiff_Ges{I}:=Sqrt(n_DefWobj_Diff_X{I}*n_DefWobj_Diff_X{I}+n_DefWobj_Diff_Y{I}*n_DefWobj_Diff_Y{I}+n_DefWobj_Diff_Z{I}*n_DefWobj_Diff_Z{I});
ENDFOR

Message:
TPErase;

TEST n_sp
CASE 1:
	TPWrite "Calculated Work Object Error(in mm) ";
	TPWrite " ";
	TPWrite "In Mess-Point 1: "\Num:=n_DefWob_jDiff_Ges{1};
	TPWrite "In Mess-Point 2: "\Num:=n_DefWob_jDiff_Ges{2};
	TPWrite "In Mess-Point 3: "\Num:=n_DefWob_jDiff_Ges{3};
	TPWrite " ";
	TPReadFK n_key,"Accept the error deviation?","No","","Info","","Yes";
CASE 2:
	TPWrite "Fehler in mm mit ermitteltem Werkobjekt";
	TPWrite " ";
	TPWrite "am Mess-Punkt 1: "\Num:=n_DefWob_jDiff_Ges{1};
	TPWrite "am Mess-Punkt 2: "\Num:=n_DefWob_jDiff_Ges{2};
	TPWrite "am Mess-Punkt 3: "\Num:=n_DefWob_jDiff_Ges{3};
	TPWrite " ";
	TPReadFK n_key,"Wird Abweichung akzeptiert?","Nein","","Info","","Ja";
CASE 3:

ENDTEST

TEST n_key
CASE 1:
	Wobj_New:=wobj_DefWobj_ACT_wobj;
	GOTO EXIT_Ende;
CASE 3:
	TPErase;

	TEST n_sp
	CASE 1:
		TPWrite "Error!! check the following:";
		TPWrite "- Incorrect/Inaccurate Measurement-Tool";
		TPWrite "- False/Inaccurate Co-ordinates ";
		TPWrite "- Incorrectly calibrated Robot";
		TPReadFK n_key,"Error > 5 mm not accepted!","","","","","OK";
	CASE 2:
	     TPWrite "Grosse Fehler können entsehen durch:";
		TPWrite "- Falsches/ungenaues Mess-Tool";
		TPWrite "- Falsche/ungenaue Koordinaten ";
		TPWrite "- unsauber geteachte Mess-Punkte";
		TPWrite "- falsch kalibrierter Roboter";
		TPReadFK n_key,"Fehler > 5 mm nicht akzeptierten!","","","","","OK";
	CASE 3:

	ENDTEST

	GOTO Message;
CASE 5:
	Wobj_New:=wobj_DefWobj_car0;
	TPErase;

	TEST n_sp
	CASE 1:
		TPWrite "The Work Object "+s_DefWobj_Wobj_Name+" was";
		TPWrite "configured correctly and ";
		TPWrite "has been stored!";
	CASE 2:
		TPWrite "Das Werkobjekt "+s_DefWobj_Wobj_Name+" wurde mit";
		TPWrite "angegebener Genauigkeit ermittelt";
		TPWrite "und gespeichert!";
	CASE 3:

	ENDTEST

	TPReadFK n_key,"","","","","","OK";

DEFAULT:
  GOTO Message;
ENDTEST

Ende:
TPErase;
EXIT;
Exit_Ende:
TPErase;
TPWrite " ";
TPWrite " ";

TEST n_sp
CASE 1:
	TPWrite "     Measurement was aborted!      ";
CASE 2:
    TPWrite "     Vermessung wurde abgebrochen!      ";
CASE 3:

ENDTEST

WaitTime 3;

ERROR
!** Error Handler **
TEST n_ErrorCode
CASE 1:
	TPErase;

	TEST n_sp
	CASE 1:
		TPWrite "Stored position";
		TPWrite "is not correct!";
	CASE 2:
		TPWrite "Gespeicherte Position kann";
		TPWrite "nicht angefahren werden!";
	CASE 3:

	ENDTEST

  	TPReadFK n_key,"","","","","","OK";
  	TRYNEXT;
CASE 2:
	M_Errror:=TRUE;

	TPErase;

	TEST n_sp
	CASE 1:
		TPWrite "The Work Object";
		TPWrite "cannot defined with the ";
		TPWrite "data entered!";
	CASE 2:
		TPWrite "Werkobjekt kann mit den";
		TPWrite "angegebenen Daten nicht";
		TPWrite "ermittelt werden!";
	CASE 3:

	ENDTEST

  	TPReadFK n_key,"","","","","","OK";
  	TRYNEXT;
DEFAULT:
  EXIT;
ENDTEST

ENDPROC !(Indirect_WOBJ)

!***************************************************************************

PROC SetHomeColl (\Num Home_Nr, \Num Collision_Nr,\String Collision_Desc)
!*************************************
!* User Routine to set collison zone *
!*        from Initproduction        *
!" When robot is in a Home position  *
!*************************************
!Home_nr            = Home position which collision zone to be requested
!Collision_Nr       = Collision zone to be requested
!Collision_Desc     = Description of other robot/s also using this collision zone

VAR string st_alias;
VAR signaldo do_TempHome;
VAR robtarget rt_CurrentPos;

CheckValue Home_Nr,1,5,0,"Home Number";
CheckValue Collision_Nr,1,62,0,"Collizone Number";

!Create signal to check home output
st_alias :="SYS_do_Home_" +NumToStr(Home_Nr,0);
AliasIO st_alias, do_TempHome;

!check if robot is in Home position and collsion zone not already occupied
IF DOutput (do_TempHome)=1 AND b_CollZoneOccupied{Collision_Nr}=FALSE THEN
	t_Home := CTool();
	wobj_home := CWobj();
	rt_CurrentPos:=CRobT(\Tool:=t_Home\WObj:=wobj_home);
	MoveJ_CollReq Collision_Nr,  rt_CurrentPos,  V10,  fine,  t_Home \ Wobj:=wobj_home\Coll_Desc:=Collision_Desc;
ENDIF

ENDPROC !(SetHomeColl)

ENDMODULE
